TYPE stRoomData :
STRUCT
	{attribute addProperty Name "<#Actual room temperature °C#>"}
	Temperature : REAL;
	{attribute addProperty Name "<#Actual room humidity %#>"}
	Humidity : REAL;
	{attribute addProperty Name "<#Actual room VOC %#>"}
	VOC : REAL;
	{attribute addProperty Name "<#Actual room CO2 concentration ppm#>"}
	CO2 : REAL;
END_STRUCT
END_TYPE

(* stored: Version 1.1.0.1, ProductVersion 3.1.4024.2
   DUT stRoomData: Id {38dbd490-63c5-420a-8bd7-131c8dfcb376} *)
